// TIA Portal project "10_Seperation_Station" (V19)

(* hardware
DEVICE "S7-1500/ET200MP station_1"  S7-1500 station
   slot 0: "Rail_0"  Rack  6ES7 590-1***0-0AA0
   slot 1: "PLC_1"  CPU 1513-1 PN  6ES7 513-1AL02-0AB0  V2.9
      slot 3: "CPU display_1"  6ES7591-1AA00-0AA0
      slot 32768: "PROFINET interface_1"  X1
         slot 32769: "Port_1"  X1 P1
         slot 32770: "Port_2"  X1 P2
      slot 34817: "Virtual CP interface port_1"  Virtual CP interface port  Virtual CP interface port
*)

// ===== PLC "PLC_1"  CPU 1513-1 PN =====

VAR_GLOBAL   // PLC tag table "Default tag table"
   "Network 2" AT %M0.0 : Bool;
   "Network 3 2nd memory" AT %M7.6 : Bool;
   "Network 3 1st memory" AT %M0.1 : Bool;
   "Network 4 1st SR GB" AT %M0.2 : Bool;
   "Network 4 2nd SR BG" AT %M1.7 : Bool;
   "M1.7 to reset M0.2 GB" AT %M2.5 : Bool;
   "Network 4 3rd SR BB" AT %M2.0 : Bool;
   "M2.0 to reset M0.2 GB" AT %M2.6 : Bool;
   "Network 4 4th SR GG" AT %M2.1 : Bool;
   "M2.1 to reset M0.2 GB" AT %M2.7 : Bool;
   "M0.2 to reset M1.7 BG" AT %M2.4 : Bool;
   "M2.0 to reset M1.7 BG" AT %M3.0 : Bool;
   "M2.1 to reset M1.7 BG" AT %M3.1 : Bool;
   "M0.2 to reset M2.0 BB" AT %M3.2 : Bool;
   "M1.7 to reset M2.0 BB" AT %M3.3 : Bool;
   "M2.1 to reset M2.0 BB" AT %M3.4 : Bool;
   "M5.1 to reset M2.1 GG" AT %M5.1 : Bool;
   "M5.2 to reset M2.1 GG" AT %M5.2 : Bool;
   "M5.3 to reset M2.1 GG" AT %M5.3 : Bool;
   "Network 13 count blue" AT %M7.4 : Bool;
   "Network 13 count green" AT %M7.5 : Bool;
   "Network 9 ap2e ec1" AT %M0.7 : Bool;
   "nw9 ec1" AT %M0.3 : Bool;
   "nw9 s1 n ec1" AT %M1.6 : Bool;
   "nw9 s1 p c1" AT %M0.4 : Bool;
   "nw9 c1" AT %M0.6 : Bool;
   "nw9 s1 n c1" AT %M0.5 : Bool;
   "nw9 c2" AT %M1.2 : Bool;
   "nw9 ec2" AT %M1.0 : Bool;
   "nw9 ap2e n c2" AT %M1.1 : Bool;
   "nw9 s1 n p1" AT %M1.3 : Bool;
   "nw9 p1" AT %M1.4 : Bool;
   "nw9 ret" AT %M1.5 : Bool;
   "nw10 ap1e ec1 ec2" AT %M7.3 : Bool;
   "nw10 s1 n" AT %M7.1 : Bool;
   "nw10 s1 p" AT %M6.7 : Bool;
   "nw10 ap1e n c1 c2" AT %M7.2 : Bool;
   "nw10 ret" AT %M2.3 : Bool;
   "nw10 SR ec1 ec2" AT %M2.2 : Bool;
   "nw10 SR c1 c2" AT %M7.0 : Bool;
   "nw11 ec1" AT %M3.6 : Bool;
   "nw11 ap1e n" AT %M4.7 : Bool;
   "nw11 c1" AT %M3.7 : Bool;
   "nw11 ec2" AT %M4.0 : Bool;
   "nw11 ap1e n ec1" AT %M5.0 : Bool;
   "nw11 s2 n" AT %M4.3 : Bool;
   "nw11 s2 p" AT %M4.4 : Bool;
   "nw11 c2" AT %M4.1 : Bool;
   "nw11 s2 n c2" AT %M4.5 : Bool;
   "nw11 p2" AT %M4.2 : Bool;
   "nw11 s2 n p2" AT %M4.6 : Bool;
   "nw11 ret" AT %M3.5 : Bool;
   "nw12 ec1" AT %M5.4 : Bool;
   "nw12 ap2e n ec1" AT %M6.6 : Bool;
   "nw12 s1 n ec1" AT %M6.2 : Bool;
   "nw12 c1" AT %M5.5 : Bool;
   "nw12 s1 p" AT %M6.1 : Bool;
   "nw12 s1 n c1" AT %M6.3 : Bool;
   "nw12 ec2" AT %M5.6 : Bool;
   "nw12 c2" AT %M5.7 : Bool;
   "nw12 ap2e n" AT %M6.5 : Bool;
   "nw12 s1 n p1" AT %M6.4 : Bool;
   "nw12 p1" AT %M6.0 : Bool;
   "nw12 ret" AT %M7.7 : Bool;
END_VAR

VAR_GLOBAL   // PLC tag table "Tag table from XML_1"
   "Start" AT %I0.0 : Bool;
   "pause and unpause" AT %I0.1 : Bool;
   "Reset" AT %I0.2 : Bool;
   "Pusher 1 front" AT %I0.3 : Bool;
   "Pusher 2 front" AT %I0.4 : Bool;
   "Pusher 1 back" AT %I0.5 : Bool;
   "Pusher 2 back" AT %I0.6 : Bool;
   "At pusher 1 exit" AT %I0.7 : Bool;
   "At pusher 2 exit" AT %I1.0 : Bool;
   "Sensor 1" AT %I1.1 : Bool;
   "Sensor 2" AT %I1.2 : Bool;
   "Start light" AT %Q0.0 : Bool;
   "P & UP light" AT %Q0.1 : Bool;
   "Reset light" AT %Q0.2 : Bool;
   "Conveyor 1" AT %Q0.3 : Bool;
   "Conveyor 2" AT %Q0.4 : Bool;
   "Entry conveyor 1" AT %Q0.5 : Bool;
   "Entry conveyor 2" AT %Q0.6 : Bool;
   "Pusher 1" AT %Q0.7 : Bool;
   "Pusher 2" AT %Q1.0 : Bool;
   "Vision sensor 1" AT %ID30 : DInt;
   "Vision sensor 2" AT %ID34 : DInt;
   "Blue Count" AT %QD30 : DInt;
   "Green Count" AT %QD34 : DInt;
END_VAR

// folder: System blocks/Program resources

DATA_BLOCK "IEC_Counter_0_DB"   // DB1
{ S7_Optimized_Access := 'TRUE' }
AUTHOR : Simatic
FAMILY : IEC
NAME : CNTR
VERSION : 1.0
// stored: InstanceOfName IEC_COUNTER
"IEC_COUNTER"
BEGIN
END_DATA_BLOCK

DATA_BLOCK "IEC_Counter_0_DB_1"   // DB2
{ S7_Optimized_Access := 'TRUE' }
AUTHOR : Simatic
FAMILY : IEC
NAME : CNTR
VERSION : 1.0
// stored: InstanceOfName IEC_COUNTER
"IEC_COUNTER"
BEGIN
END_DATA_BLOCK

// folder: (top level)

ORGANIZATION_BLOCK "Main"   // OB1, LAD, ProgramCycle
TITLE = "Main Program Sweep (Cycle)"
{ S7_Optimized_Access := 'TRUE' }
VERSION : 0.1
   VAR_INPUT
      Initial_Call : Bool;   // Initial call of this OB
      Remanence : Bool;   // =True, if remanent data are available
   END_VAR
   VAR_TEMP   // added for the SCL form of the ladder/FBD networks
      _w1 : Bool;
      _w2 : Bool;
      _w3 : Bool;
      _w4 : Bool;
      _w5 : Bool;
      _w6 : Bool;
      _w7 : Bool;
      _w8 : Bool;
      _w9 : Bool;
      _w10 : Bool;
      _w11 : Bool;
      _w12 : Bool;
      _w13 : Bool;
      _w14 : Bool;
   END_VAR
BEGIN

REGION Network 2: Start Reset system with ON/OFF LEDs
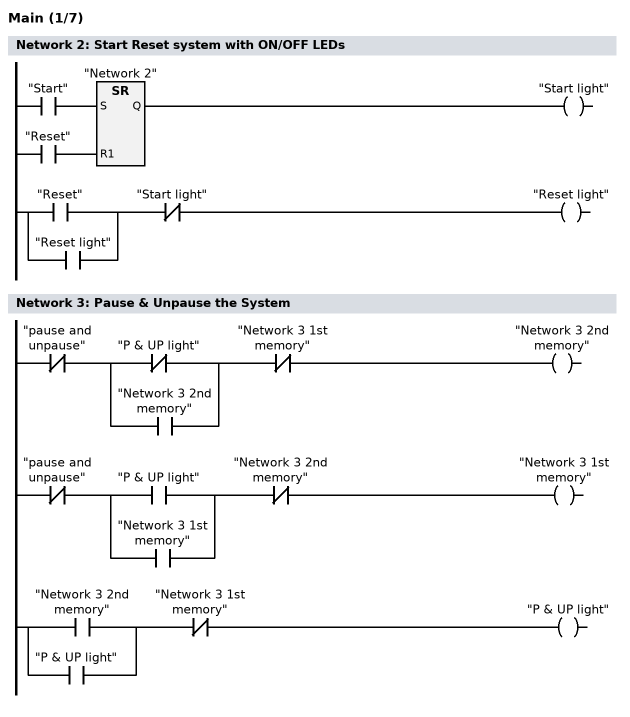
   RUNG wire#powerrail
      Contact( "Start" )
      S_SR(operand := "Network 2", r1 := wire#w1)
      Coil( "Start light" )
   END_RUNG
   RUNG wire#powerrail
      Contact( "Reset" )
   END_RUNG wire#w1
   RUNG wire#powerrail
      Contact( "Reset" )
      wire#w2
      I_Contact( "Start light" )
      Coil( "Reset light" )
   END_RUNG
   RUNG wire#powerrail
      Contact( "Reset light" )
   END_RUNG wire#w2
   // the same network as SCL:
   IF "Start" THEN
       "Network 2" := TRUE;   // SR flip-flop
   END_IF;
   IF "Reset" THEN "Network 2" := FALSE; END_IF;
   "Start light" := "Network 2";
   "Reset light" := ("Reset" OR "Reset light") AND NOT "Start light";
END_REGION

REGION Network 3: Pause & Unpause the System
   RUNG wire#powerrail
      I_Contact( "pause and unpause" )
      wire#w1
      I_Contact( "P & UP light" )
      wire#w2
      I_Contact( "Network 3 1st memory" )
      Coil( "Network 3 2nd memory" )
   END_RUNG
   RUNG wire#w1
      Contact( "Network 3 2nd memory" )
   END_RUNG wire#w2
   RUNG wire#powerrail
      I_Contact( "pause and unpause" )
      wire#w3
      Contact( "P & UP light" )
      wire#w4
      I_Contact( "Network 3 2nd memory" )
      Coil( "Network 3 1st memory" )
   END_RUNG
   RUNG wire#w3
      Contact( "Network 3 1st memory" )
   END_RUNG wire#w4
   RUNG wire#powerrail
      Contact( "Network 3 2nd memory" )
      wire#w5
      I_Contact( "Network 3 1st memory" )
      Coil( "P & UP light" )
   END_RUNG
   RUNG wire#powerrail
      Contact( "P & UP light" )
   END_RUNG wire#w5
   // the same network as SCL:
   "Network 3 2nd memory" := NOT "pause and unpause" AND (NOT "P & UP light" OR "Network 3 2nd memory") AND NOT "Network 3 1st memory";
   "Network 3 1st memory" := NOT "pause and unpause" AND ("P & UP light" OR "Network 3 1st memory") AND NOT "Network 3 2nd memory";
   "P & UP light" := ("Network 3 2nd memory" OR "P & UP light") AND NOT "Network 3 1st memory";
END_REGION

REGION Network 4: We have 2 vision sensor and 2 color, we will divide it to 4 cases
   // Sensor = 4 means green, sensor = 1 means blue
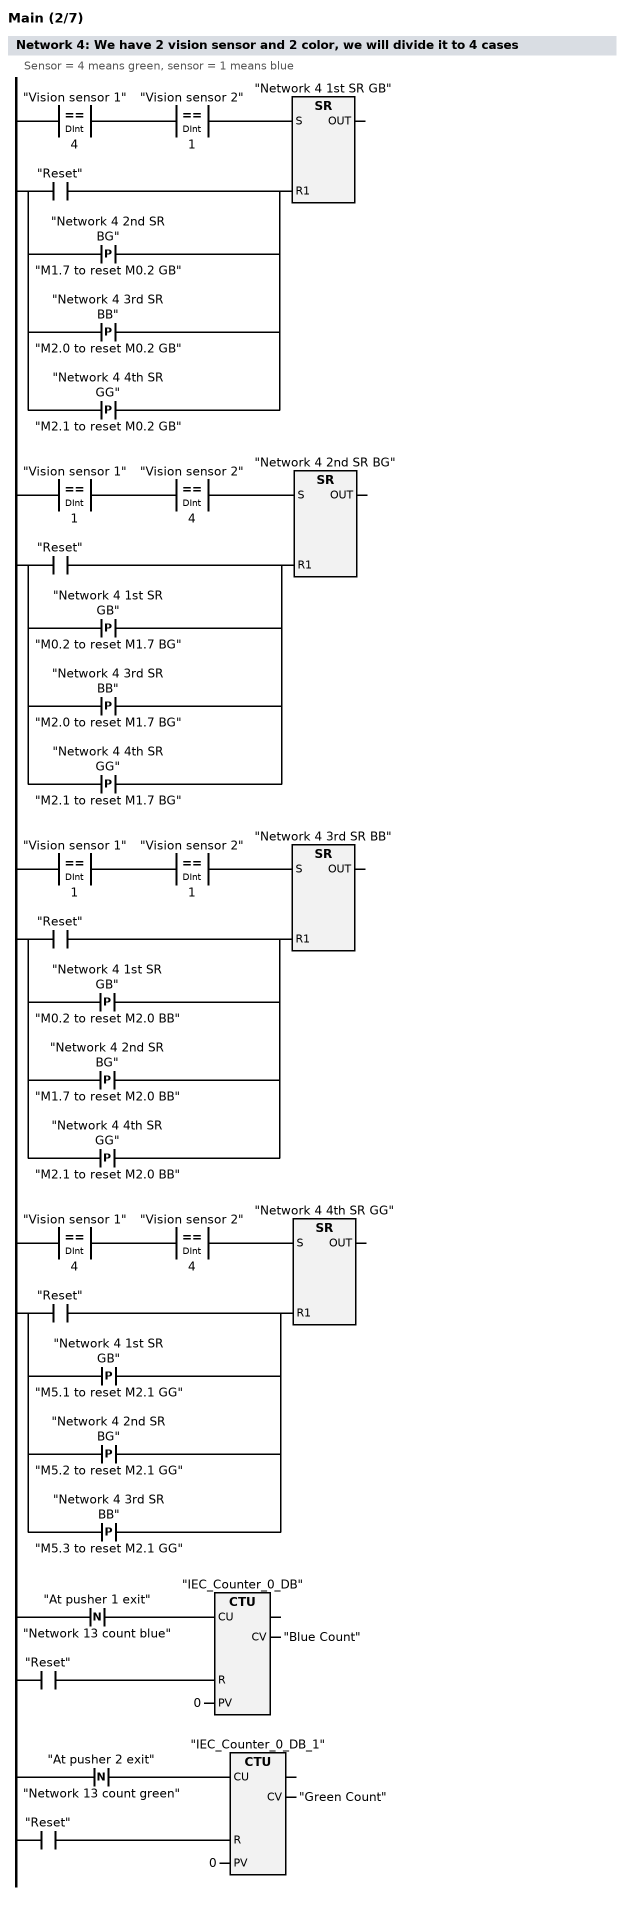
   #_w1 := "Network 4 2nd SR BG" AND NOT "M1.7 to reset M0.2 GB";   // rising edge of "Network 4 2nd SR BG"
   "M1.7 to reset M0.2 GB" := "Network 4 2nd SR BG";
   #_w2 := "Network 4 3rd SR BB" AND NOT "M2.0 to reset M0.2 GB";   // rising edge of "Network 4 3rd SR BB"
   "M2.0 to reset M0.2 GB" := "Network 4 3rd SR BB";
   #_w3 := "Network 4 4th SR GG" AND NOT "M2.1 to reset M0.2 GB";   // rising edge of "Network 4 4th SR GG"
   "M2.1 to reset M0.2 GB" := "Network 4 4th SR GG";
   IF ("Vision sensor 1" = 4) AND ("Vision sensor 2" = 1) THEN
       "Network 4 1st SR GB" := TRUE;   // SR flip-flop
   END_IF;
   IF "Reset" OR #_w1 OR #_w2 OR #_w3 THEN "Network 4 1st SR GB" := FALSE; END_IF;
   #_w4 := "Network 4 1st SR GB" AND NOT "M0.2 to reset M1.7 BG";   // rising edge of "Network 4 1st SR GB"
   "M0.2 to reset M1.7 BG" := "Network 4 1st SR GB";
   #_w5 := "Network 4 3rd SR BB" AND NOT "M2.0 to reset M1.7 BG";   // rising edge of "Network 4 3rd SR BB"
   "M2.0 to reset M1.7 BG" := "Network 4 3rd SR BB";
   #_w6 := "Network 4 4th SR GG" AND NOT "M2.1 to reset M1.7 BG";   // rising edge of "Network 4 4th SR GG"
   "M2.1 to reset M1.7 BG" := "Network 4 4th SR GG";
   IF ("Vision sensor 1" = 1) AND ("Vision sensor 2" = 4) THEN
       "Network 4 2nd SR BG" := TRUE;   // SR flip-flop
   END_IF;
   IF "Reset" OR #_w4 OR #_w5 OR #_w6 THEN "Network 4 2nd SR BG" := FALSE; END_IF;
   #_w7 := "Network 4 1st SR GB" AND NOT "M0.2 to reset M2.0 BB";   // rising edge of "Network 4 1st SR GB"
   "M0.2 to reset M2.0 BB" := "Network 4 1st SR GB";
   #_w8 := "Network 4 2nd SR BG" AND NOT "M1.7 to reset M2.0 BB";   // rising edge of "Network 4 2nd SR BG"
   "M1.7 to reset M2.0 BB" := "Network 4 2nd SR BG";
   #_w9 := "Network 4 4th SR GG" AND NOT "M2.1 to reset M2.0 BB";   // rising edge of "Network 4 4th SR GG"
   "M2.1 to reset M2.0 BB" := "Network 4 4th SR GG";
   IF ("Vision sensor 1" = 1) AND ("Vision sensor 2" = 1) THEN
       "Network 4 3rd SR BB" := TRUE;   // SR flip-flop
   END_IF;
   IF "Reset" OR #_w7 OR #_w8 OR #_w9 THEN "Network 4 3rd SR BB" := FALSE; END_IF;
   #_w10 := "Network 4 1st SR GB" AND NOT "M5.1 to reset M2.1 GG";   // rising edge of "Network 4 1st SR GB"
   "M5.1 to reset M2.1 GG" := "Network 4 1st SR GB";
   #_w11 := "Network 4 2nd SR BG" AND NOT "M5.2 to reset M2.1 GG";   // rising edge of "Network 4 2nd SR BG"
   "M5.2 to reset M2.1 GG" := "Network 4 2nd SR BG";
   #_w12 := "Network 4 3rd SR BB" AND NOT "M5.3 to reset M2.1 GG";   // rising edge of "Network 4 3rd SR BB"
   "M5.3 to reset M2.1 GG" := "Network 4 3rd SR BB";
   IF ("Vision sensor 1" = 4) AND ("Vision sensor 2" = 4) THEN
       "Network 4 4th SR GG" := TRUE;   // SR flip-flop
   END_IF;
   IF "Reset" OR #_w10 OR #_w11 OR #_w12 THEN "Network 4 4th SR GG" := FALSE; END_IF;
   #_w13 := NOT "At pusher 1 exit" AND "Network 13 count blue";   // falling edge of "At pusher 1 exit"
   "Network 13 count blue" := "At pusher 1 exit";
   "IEC_Counter_0_DB".CTU(CU := #_w13, R := "Reset", PV := 0, CV => "Blue Count");
   #_w14 := NOT "At pusher 2 exit" AND "Network 13 count green";   // falling edge of "At pusher 2 exit"
   "Network 13 count green" := "At pusher 2 exit";
   "IEC_Counter_0_DB_1".CTU(CU := #_w14, R := "Reset", PV := 0, CV => "Green Count");
END_REGION

REGION Network 5: To activate Network 9 immediatly
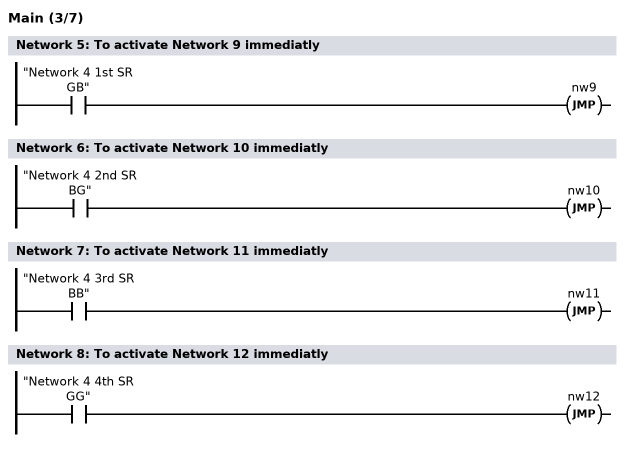
   RUNG wire#powerrail
      Contact( "Network 4 1st SR GB" )
      JumpCoil( nw9 )
   END_RUNG
   // the same network as SCL:
   IF "Network 4 1st SR GB" THEN GOTO nw9; END_IF;
END_REGION

REGION Network 6: To activate Network 10 immediatly
   RUNG wire#powerrail
      Contact( "Network 4 2nd SR BG" )
      JumpCoil( nw10 )
   END_RUNG
   // the same network as SCL:
   IF "Network 4 2nd SR BG" THEN GOTO nw10; END_IF;
END_REGION

REGION Network 7: To activate Network 11 immediatly
   RUNG wire#powerrail
      Contact( "Network 4 3rd SR BB" )
      JumpCoil( nw11 )
   END_RUNG
   // the same network as SCL:
   IF "Network 4 3rd SR BB" THEN GOTO nw11; END_IF;
END_REGION

REGION Network 8: To activate Network 12 immediatly
   RUNG wire#powerrail
      Contact( "Network 4 4th SR GG" )
      JumpCoil( nw12 )
   END_RUNG
   // the same network as SCL:
   IF "Network 4 4th SR GG" THEN GOTO nw12; END_IF;
END_REGION

REGION Network 9: Green on Conveyor 1 and Blue on conveyor 2
   // Pusher 1 move green from 1st conveyor to 2nd conveyor
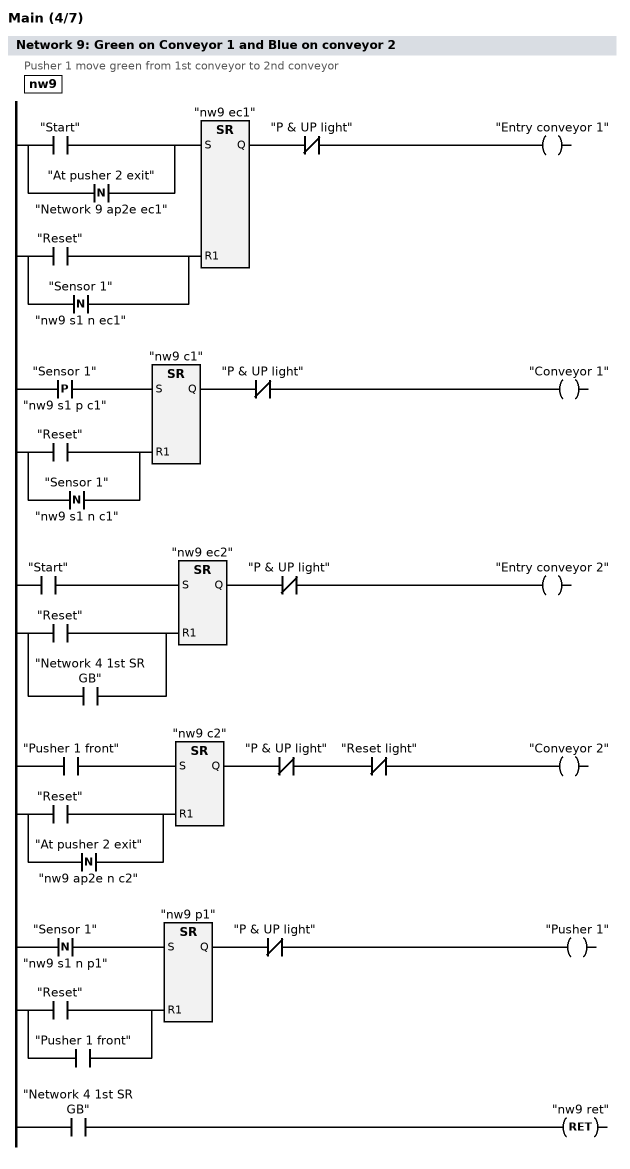
   nw9:
   #_w1 := NOT "At pusher 2 exit" AND "Network 9 ap2e ec1";   // falling edge of "At pusher 2 exit"
   "Network 9 ap2e ec1" := "At pusher 2 exit";
   #_w2 := NOT "Sensor 1" AND "nw9 s1 n ec1";   // falling edge of "Sensor 1"
   "nw9 s1 n ec1" := "Sensor 1";
   IF "Start" OR #_w1 THEN
       "nw9 ec1" := TRUE;   // SR flip-flop
   END_IF;
   IF "Reset" OR #_w2 THEN "nw9 ec1" := FALSE; END_IF;
   "Entry conveyor 1" := "nw9 ec1" AND NOT "P & UP light";
   #_w3 := "Sensor 1" AND NOT "nw9 s1 p c1";   // rising edge of "Sensor 1"
   "nw9 s1 p c1" := "Sensor 1";
   #_w4 := NOT "Sensor 1" AND "nw9 s1 n c1";   // falling edge of "Sensor 1"
   "nw9 s1 n c1" := "Sensor 1";
   IF #_w3 THEN
       "nw9 c1" := TRUE;   // SR flip-flop
   END_IF;
   IF "Reset" OR #_w4 THEN "nw9 c1" := FALSE; END_IF;
   "Conveyor 1" := "nw9 c1" AND NOT "P & UP light";
   IF "Start" THEN
       "nw9 ec2" := TRUE;   // SR flip-flop
   END_IF;
   IF "Reset" OR "Network 4 1st SR GB" THEN "nw9 ec2" := FALSE; END_IF;
   "Entry conveyor 2" := "nw9 ec2" AND NOT "P & UP light";
   #_w5 := NOT "At pusher 2 exit" AND "nw9 ap2e n c2";   // falling edge of "At pusher 2 exit"
   "nw9 ap2e n c2" := "At pusher 2 exit";
   IF "Pusher 1 front" THEN
       "nw9 c2" := TRUE;   // SR flip-flop
   END_IF;
   IF "Reset" OR #_w5 THEN "nw9 c2" := FALSE; END_IF;
   "Conveyor 2" := "nw9 c2" AND NOT "P & UP light" AND NOT "Reset light";
   #_w6 := NOT "Sensor 1" AND "nw9 s1 n p1";   // falling edge of "Sensor 1"
   "nw9 s1 n p1" := "Sensor 1";
   IF #_w6 THEN
       "nw9 p1" := TRUE;   // SR flip-flop
   END_IF;
   IF "Reset" OR "Pusher 1 front" THEN "nw9 p1" := FALSE; END_IF;
   "Pusher 1" := "nw9 p1" AND NOT "P & UP light";
   IF "Network 4 1st SR GB" THEN
       ENO := "nw9 ret";
       RETURN;
   END_IF;
END_REGION

REGION Network 10: Green on Conveyor 2 & Blue on Conveyor 1 (dont need to sperate)
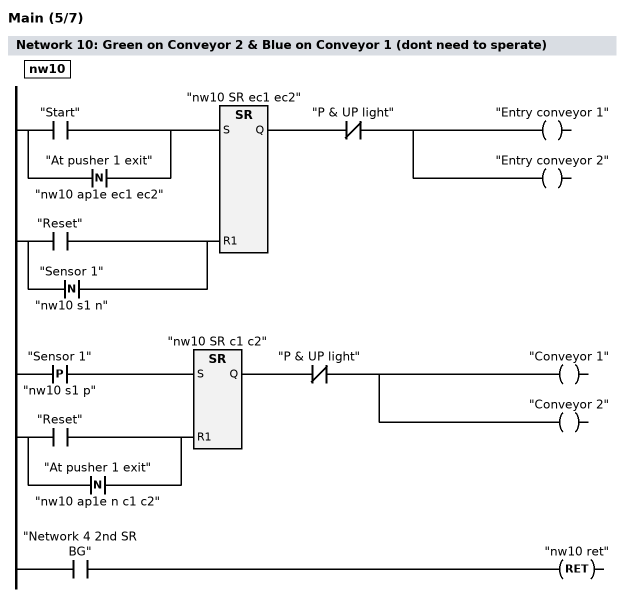
   nw10:
   #_w1 := NOT "At pusher 1 exit" AND "nw10 ap1e ec1 ec2";   // falling edge of "At pusher 1 exit"
   "nw10 ap1e ec1 ec2" := "At pusher 1 exit";
   #_w2 := NOT "Sensor 1" AND "nw10 s1 n";   // falling edge of "Sensor 1"
   "nw10 s1 n" := "Sensor 1";
   IF "Start" OR #_w1 THEN
       "nw10 SR ec1 ec2" := TRUE;   // SR flip-flop
   END_IF;
   IF "Reset" OR #_w2 THEN "nw10 SR ec1 ec2" := FALSE; END_IF;
   "Entry conveyor 1" := "nw10 SR ec1 ec2" AND NOT "P & UP light";
   "Entry conveyor 2" := "Entry conveyor 1";
   #_w3 := "Sensor 1" AND NOT "nw10 s1 p";   // rising edge of "Sensor 1"
   "nw10 s1 p" := "Sensor 1";
   #_w4 := NOT "At pusher 1 exit" AND "nw10 ap1e n c1 c2";   // falling edge of "At pusher 1 exit"
   "nw10 ap1e n c1 c2" := "At pusher 1 exit";
   IF #_w3 THEN
       "nw10 SR c1 c2" := TRUE;   // SR flip-flop
   END_IF;
   IF "Reset" OR #_w4 THEN "nw10 SR c1 c2" := FALSE; END_IF;
   "Conveyor 1" := "nw10 SR c1 c2" AND NOT "P & UP light";
   "Conveyor 2" := "Conveyor 1";
   IF "Network 4 2nd SR BG" THEN
       ENO := "nw10 ret";
       RETURN;
   END_IF;
END_REGION

REGION Network 11: Blue on conveyor 1 & 2 (Pusher 2 moves blue from 2nd conveyor to 1st conveyor)
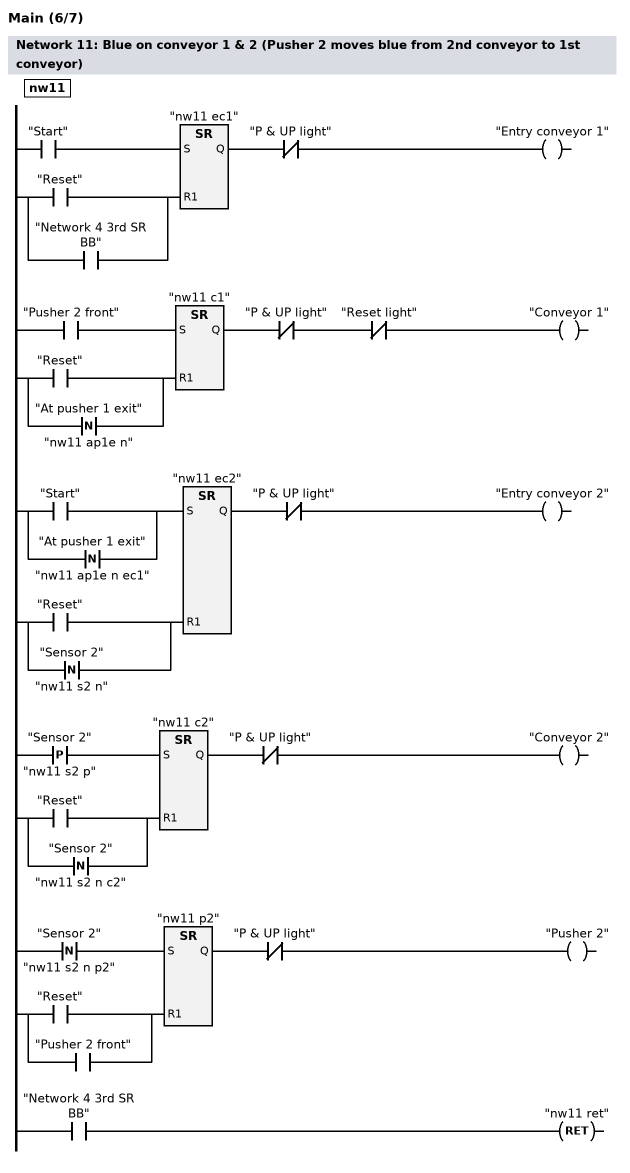
   nw11:
   IF "Start" THEN
       "nw11 ec1" := TRUE;   // SR flip-flop
   END_IF;
   IF "Reset" OR "Network 4 3rd SR BB" THEN "nw11 ec1" := FALSE; END_IF;
   "Entry conveyor 1" := "nw11 ec1" AND NOT "P & UP light";
   #_w1 := NOT "At pusher 1 exit" AND "nw11 ap1e n";   // falling edge of "At pusher 1 exit"
   "nw11 ap1e n" := "At pusher 1 exit";
   IF "Pusher 2 front" THEN
       "nw11 c1" := TRUE;   // SR flip-flop
   END_IF;
   IF "Reset" OR #_w1 THEN "nw11 c1" := FALSE; END_IF;
   "Conveyor 1" := "nw11 c1" AND NOT "P & UP light" AND NOT "Reset light";
   #_w2 := NOT "At pusher 1 exit" AND "nw11 ap1e n ec1";   // falling edge of "At pusher 1 exit"
   "nw11 ap1e n ec1" := "At pusher 1 exit";
   #_w3 := NOT "Sensor 2" AND "nw11 s2 n";   // falling edge of "Sensor 2"
   "nw11 s2 n" := "Sensor 2";
   IF "Start" OR #_w2 THEN
       "nw11 ec2" := TRUE;   // SR flip-flop
   END_IF;
   IF "Reset" OR #_w3 THEN "nw11 ec2" := FALSE; END_IF;
   "Entry conveyor 2" := "nw11 ec2" AND NOT "P & UP light";
   #_w4 := "Sensor 2" AND NOT "nw11 s2 p";   // rising edge of "Sensor 2"
   "nw11 s2 p" := "Sensor 2";
   #_w5 := NOT "Sensor 2" AND "nw11 s2 n c2";   // falling edge of "Sensor 2"
   "nw11 s2 n c2" := "Sensor 2";
   IF #_w4 THEN
       "nw11 c2" := TRUE;   // SR flip-flop
   END_IF;
   IF "Reset" OR #_w5 THEN "nw11 c2" := FALSE; END_IF;
   "Conveyor 2" := "nw11 c2" AND NOT "P & UP light";
   #_w6 := NOT "Sensor 2" AND "nw11 s2 n p2";   // falling edge of "Sensor 2"
   "nw11 s2 n p2" := "Sensor 2";
   IF #_w6 THEN
       "nw11 p2" := TRUE;   // SR flip-flop
   END_IF;
   IF "Reset" OR "Pusher 2 front" THEN "nw11 p2" := FALSE; END_IF;
   "Pusher 2" := "nw11 p2" AND NOT "P & UP light";
   IF "Network 4 3rd SR BB" THEN
       ENO := "nw11 ret";
       RETURN;
   END_IF;
END_REGION

REGION Network 12: Green Conveyor 1 & 2
   // Pusher 1 moves green from 1st conveyor to 2nd
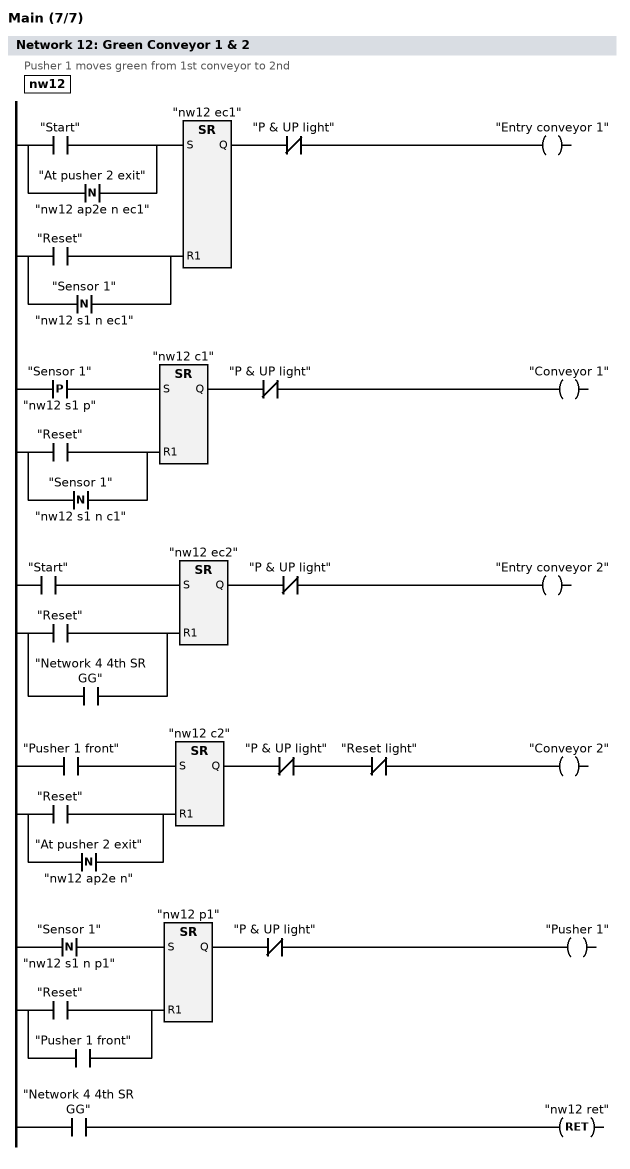
   nw12:
   #_w1 := NOT "At pusher 2 exit" AND "nw12 ap2e n ec1";   // falling edge of "At pusher 2 exit"
   "nw12 ap2e n ec1" := "At pusher 2 exit";
   #_w2 := NOT "Sensor 1" AND "nw12 s1 n ec1";   // falling edge of "Sensor 1"
   "nw12 s1 n ec1" := "Sensor 1";
   IF "Start" OR #_w1 THEN
       "nw12 ec1" := TRUE;   // SR flip-flop
   END_IF;
   IF "Reset" OR #_w2 THEN "nw12 ec1" := FALSE; END_IF;
   "Entry conveyor 1" := "nw12 ec1" AND NOT "P & UP light";
   #_w3 := "Sensor 1" AND NOT "nw12 s1 p";   // rising edge of "Sensor 1"
   "nw12 s1 p" := "Sensor 1";
   #_w4 := NOT "Sensor 1" AND "nw12 s1 n c1";   // falling edge of "Sensor 1"
   "nw12 s1 n c1" := "Sensor 1";
   IF #_w3 THEN
       "nw12 c1" := TRUE;   // SR flip-flop
   END_IF;
   IF "Reset" OR #_w4 THEN "nw12 c1" := FALSE; END_IF;
   "Conveyor 1" := "nw12 c1" AND NOT "P & UP light";
   IF "Start" THEN
       "nw12 ec2" := TRUE;   // SR flip-flop
   END_IF;
   IF "Reset" OR "Network 4 4th SR GG" THEN "nw12 ec2" := FALSE; END_IF;
   "Entry conveyor 2" := "nw12 ec2" AND NOT "P & UP light";
   #_w5 := NOT "At pusher 2 exit" AND "nw12 ap2e n";   // falling edge of "At pusher 2 exit"
   "nw12 ap2e n" := "At pusher 2 exit";
   IF "Pusher 1 front" THEN
       "nw12 c2" := TRUE;   // SR flip-flop
   END_IF;
   IF "Reset" OR #_w5 THEN "nw12 c2" := FALSE; END_IF;
   "Conveyor 2" := "nw12 c2" AND NOT "P & UP light" AND NOT "Reset light";
   #_w6 := NOT "Sensor 1" AND "nw12 s1 n p1";   // falling edge of "Sensor 1"
   "nw12 s1 n p1" := "Sensor 1";
   IF #_w6 THEN
       "nw12 p1" := TRUE;   // SR flip-flop
   END_IF;
   IF "Reset" OR "Pusher 1 front" THEN "nw12 p1" := FALSE; END_IF;
   "Pusher 1" := "nw12 p1" AND NOT "P & UP light";
   IF "Network 4 4th SR GG" THEN
       ENO := "nw12 ret";
       RETURN;
   END_IF;
END_REGION
END_ORGANIZATION_BLOCK